// TIA Portal V20 export
DATA_BLOCK "DB_Alarms"   // DB300
// stored: AutoNumber false, InstanceOfName FB_Alarms, InstanceOfType FB
"FB_Alarms"
   // VAR
   //    sAlarmsLevel0 : Bool;
   //    sAlarmsLevel1 : Bool;
   //    sAlarmsLevel2 : Bool;
   //    sAlarmsLevel3 : Bool;
   //    sAlarmsLevel4 : Bool;
   //    sAlarmsLevel5 : Bool;
   //    sAlarmsLevel6 : Bool;
   //    sRTBuzzer { S7_SetPoint := 'True'} : R_TRIG;
   //    sActiveBuzzer : Bool;
   //    sTableInParkPosition : Bool;
   // END_VAR
BEGIN
END_DATA_BLOCK
